FUNCTION TryConvert_BYTE_TO_DT : BOOL
VAR_INPUT
	in : BYTE;
	out : REFERENCE TO DT;
END_VAR

out := BYTE_TO_DT(in);
TryConvert_BYTE_TO_DT := TRUE;

END_FUNCTION

(* stored: Version 1.1.0.1, ProductVersion 3.1.4024.12
   POU TryConvert_BYTE_TO_DT: Id {9d945841-5645-48b7-b067-bdd2d0e706ad}, SpecialFunc None *)
